// TIA Portal V20 export
TYPE "typeHotWireCutter"
// stored: Access Published, IsFailsafeCompliant true, Namespace Safety
   STRUCT
      on : Bool;
      off : Bool;
   END_STRUCT;
END_TYPE
